INTERFACE ITcoCodeReader EXTENDS __System.IQueryInterface

METHOD StartAtMain : TcoCore.ITcoTaskStatus
END_METHOD

METHOD StartMovements : TcoCore.ITcoTaskStatus
END_METHOD

END_INTERFACE

(* stored: Version 1.1.0.1, ProductVersion 3.1.4024.12
   Itf ITcoCodeReader: Id {20e8eca5-ad98-0994-0a1f-244ff926d52d}
   Folder Operations: Id {4433432c-54c1-0b18-0651-81d20a55bbd9}
   Method StartAtMain: Id {e6ef27be-4d76-0c9a-1cb7-1307326132ec}
   Method StartMovements: Id {3b5fd205-da52-04d1-30cf-1c3c24bc0135} *)
